// TIA Portal project "BTL_FIX" (V16)

(* hardware
DEVICE "S7300/ET200M station_1"  S7-300 station
   slot 0: "Rail_0"  Rail  6ES7 390-1***0-0AA0
   slot 2: "PLC_1"  CPU 314C-2 PN/DP  6ES7 314-6EH04-0AB0  V3.3
      slot 2: "PROFINET interface_1"  PN-IO
         slot 1: "Port_1"  Port
         slot 2: "Port_2"  Port
      slot 5: "DI 24/DO 16_1"  DI24/DO16
      slot 6: "AI 5/AO 2_1"  AI5/AO2
      slot 7: "Count_1"  Counter
      slot 8: "Positioning_1"  Positioning
   slot 4: "DO 8x24VDC/0.5A_1"  DO8 x 24VDC / 0.5A  6ES7 322-8BF00-0AB0
*)

// ===== PLC "PLC_1"  CPU 314C-2 PN/DP =====

VAR_GLOBAL   // PLC tag table "Default tag table"
   "Tag_1" AT %M100.0 : Bool;
   "Tag_2" AT %M200.0 : Bool;
   "Tag_3" AT %M201.0 : Bool;
END_VAR

VAR_GLOBAL   // PLC tag table "PRO_TAG"
   "Start" AT %I0.0 : Bool;
   "Pause" AT %I0.1 : Bool;
   "EMER" AT %I0.2 : Bool;
   "RESET" AT %I0.3 : Bool;
   "MODE" AT %I0.4 : Bool;
   "HALF_AUTO" AT %I2.6 : Bool;
   "PHOI" AT %I0.5 : Bool;
   "A0" AT %I1.0 : Bool;
   "A1" AT %I1.1 : Bool;
   "B0" AT %I1.2 : Bool;
   "B1" AT %I1.3 : Bool;
   "C0" AT %I1.4 : Bool;
   "C1" AT %I1.5 : Bool;
   "A_FOR" AT %Q0.0 : Bool;
   "A_REV" AT %Q0.1 : Bool;
   "B_FOR" AT %Q0.2 : Bool;
   "B_REV" AT %Q0.3 : Bool;
   "C_FOR" AT %Q0.4 : Bool;
   "C_REV" AT %Q0.5 : Bool;
   "S0" AT %M8.0 : Bool;
   "S1" AT %M8.1 : Bool;
   "S2" AT %M8.2 : Bool;
   "S3" AT %M8.3 : Bool;
   "S4" AT %M8.4 : Bool;
   "S5" AT %M8.5 : Bool;
   "S6" AT %M8.6 : Bool;
   "S7" AT %M8.7 : Bool;
   "S_NULL" AT %M9.0 : Bool;
   "S_EMER" AT %M9.1 : Bool;
   "S_PAUSE" AT %M9.2 : Bool;
   "T01" AT %M3.1 : Bool;
   "T1_PAUSE" AT %M3.2 : Bool;
   "T1_EMER" AT %M3.3 : Bool;
   "T12" AT %M3.4 : Bool;
   "T2_PAUSE" AT %M3.5 : Bool;
   "T2_EMER" AT %M3.6 : Bool;
   "T23" AT %M3.7 : Bool;
   "T3_PAUSE" AT %M4.0 : Bool;
   "T3_EMER" AT %M4.1 : Bool;
   "T34" AT %M4.2 : Bool;
   "T4_PAUSE" AT %M4.3 : Bool;
   "T4_EMER" AT %M4.4 : Bool;
   "T45" AT %M4.5 : Bool;
   "T5_PAUSE" AT %M4.6 : Bool;
   "T5_EMER" AT %M4.7 : Bool;
   "T56" AT %M5.0 : Bool;
   "T6_PAUSE" AT %M5.1 : Bool;
   "T6_EMER" AT %M5.2 : Bool;
   "T67" AT %M5.3 : Bool;
   "T7_PAUSE" AT %M5.4 : Bool;
   "T7_EMER" AT %M5.5 : Bool;
   "T7_NULL" AT %M5.6 : Bool;
   "T_NULL_S1" AT %M5.7 : Bool;
   "T_EMER_RESET" AT %M6.0 : Bool;
   "T_PAUSE_EMER" AT %M6.1 : Bool;
   "T_PAUSE_S1" AT %M6.2 : Bool;
   "T_PAUSE_S2" AT %M6.3 : Bool;
   "T_PAUSE_S3" AT %M6.4 : Bool;
   "T_PAUSE_S4" AT %M6.5 : Bool;
   "T_PAUSE_S5" AT %M6.6 : Bool;
   "T_PAUSE_S6" AT %M6.7 : Bool;
   "T_PAUSE_S7" AT %M7.0 : Bool;
   "T_PAUSE_NULL" AT %M7.1 : Bool;
   "T_NULL_PAUSE" AT %M7.2 : Bool;
   "T_NULL_EMER" AT %M7.3 : Bool;
   "INT_PAUSE" AT %MW10 : Int;
   "T00" AT %M3.0 : Bool;
   "TEMP_START" AT %M7.4 : Bool;
   "Q_START" AT %Q0.6 : Bool;
   "Q_MODE" AT %Q0.7 : Bool;
   "Q_WAIT" AT %Q1.6 : Bool;
   "FIRST_SCAN" AT %M1.7 : Bool;
   "TEMP_FIRST" AT %M2.0 : Bool;
   "S_RESET" AT %M2.1 : Bool;
   "T_RESET_S1" AT %M2.2 : Bool;
   "no_name" AT %M2.3 : Bool;
   "Q_EMER" AT %Q1.7 : Bool;
   "INA_FOR" AT %I2.0 : Bool;
   "INA_REV" AT %I2.1 : Bool;
   "INB_FOR" AT %I2.2 : Bool;
   "INB_REV" AT %I2.3 : Bool;
   "INC_FOR" AT %I2.4 : Bool;
   "INC_REV" AT %I2.5 : Bool;
   "Q_PAUSE" AT %Q1.0 : Bool;
   "HA_FOR" AT %M0.0 : Bool;
   "HA_REV" AT %M0.1 : Bool;
   "HB_FOR" AT %M0.2 : Bool;
   "HB_REV" AT %M0.3 : Bool;
   "HC_FOR" AT %M0.4 : Bool;
   "HC_REV" AT %M0.5 : Bool;
   "Q_PHOI" AT %Q1.1 : Bool;
   "STOP" AT %I0.6 : Bool;
   "TEMP_OFF" AT %M0.6 : Bool;
   "PHOI_MOI" AT %M200.1 : Bool;
   "T_NULL_OFF" AT %M200.2 : Bool;
   "S_OFF" AT %M200.3 : Bool;
   "T_OFF_S1" AT %M200.4 : Bool;
   "L_ERROR_PHOI" AT %Q2.0 : Bool;
   "L_OFF" AT %Q2.1 : Bool;
   "TRIG_MODE" AT %M200.5 : Bool;
   "TMP_TRIG_MODE" AT %M200.6 : Bool;
   "ALARM_AR" AT %Q2.2 : Bool;
   "ALARM_AF" AT %Q2.3 : Bool;
   "ALARM_BR" AT %Q2.4 : Bool;
   "ALARM_BF" AT %Q2.5 : Bool;
   "ALARM_CR" AT %Q2.6 : Bool;
   "ALARM_CF" AT %Q2.7 : Bool;
   "PHOI_NOT_FOUND" AT %M200.7 : Bool;
END_VAR

FUNCTION "Block_1" : Void   // FC1, LAD
{ S7_Optimized_Access := 'FALSE' }
VERSION : 0.1
   VAR_INPUT
      in : Bool;
   END_VAR
   VAR_OUTPUT
      out : Bool;
   END_VAR
   VAR_TEMP   // added for the SCL form of the ladder/FBD networks
      _w1 : Bool;
   END_VAR
BEGIN

REGION Network 1
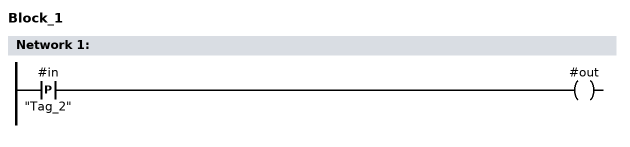
   RUNG wire#powerrail
      P_Contact(operand := #in, bit := "Tag_2")
      Coil( #out )
   END_RUNG
   // the same network as SCL:
   #_w1 := #in AND NOT "Tag_2";   // rising edge of #in
   "Tag_2" := #in;
   #out := #_w1;
END_REGION
END_FUNCTION

FUNCTION "Block_2" : Void   // FC2, LAD
{ S7_Optimized_Access := 'FALSE' }
VERSION : 0.1
   VAR_INPUT
      in : Bool;
   END_VAR
   VAR_OUTPUT
      out : Bool;
   END_VAR
   VAR_TEMP   // added for the SCL form of the ladder/FBD networks
      _w1 : Bool;
   END_VAR
BEGIN

REGION Network 1
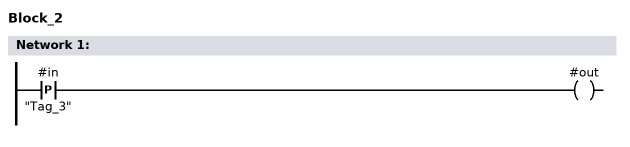
   RUNG wire#powerrail
      P_Contact(operand := #in, bit := "Tag_3")
      Coil( #out )
   END_RUNG
   // the same network as SCL:
   #_w1 := #in AND NOT "Tag_3";   // rising edge of #in
   "Tag_3" := #in;
   #out := #_w1;
END_REGION
END_FUNCTION

ORGANIZATION_BLOCK "Main"   // OB1, SCL
TITLE = "Main Program Sweep (Cycle)"
{ S7_Optimized_Access := 'FALSE' }
VERSION : 0.1
   VAR_TEMP
      OB1_EV_CLASS : Byte;   // Bits 0-3 = 1 (Coming event), Bits 4-7 = 1 (Event class 1)
      OB1_SCAN_1 : Byte;   // 1 (Cold restart scan 1 of OB 1), 3 (Scan 2-n of OB 1)
      OB1_PRIORITY : Byte;   // Priority of OB Execution
      OB1_OB_NUMBR : Byte;   // 1 (Organization block 1, OB1)
      OB1_RESERVED_1 : Byte;   // Reserved for system
      OB1_RESERVED_2 : Byte;   // Reserved for system
      OB1_PREV_CYCLE : Int;   // Cycle time of previous OB1 scan (milliseconds)
      OB1_MIN_CYCLE : Int;   // Minimum cycle time of OB1 (milliseconds)
      OB1_MAX_CYCLE : Int;   // Maximum cycle time of OB1 (milliseconds)
      OB1_DATE_TIME : Date_And_Time;   // Date and time OB1 started
   END_VAR
BEGIN
   "IEC_Timer_0_DB".TON(IN:="S_NULL",
                        PT:=T#1S);
   "IEC_Timer_0_DB_1".TOF(IN:="PHOI_MOI",
                          PT:=t#2s);

   IF "STOP" AND NOT "S_EMER" AND NOT "EMER" THEN
       "TEMP_OFF" := 1;
   END_IF;
   IF "TEMP_OFF" AND "Start" THEN
       "TEMP_OFF" := 0;
   END_IF;

   IF NOT "S_EMER" THEN
       "Block_1"(in := "MODE",
                 out => "TRIG_MODE");
   END_IF;
   "Block_2"(in:="PHOI",
             out=>"PHOI_MOI");

   REGION
       "Q_MODE" := "MODE";
       "Q_START" := "TEMP_START" AND NOT "S_EMER";
       "Q_WAIT" := "S_NULL" AND NOT "TEMP_OFF" AND "MODE";
       "Q_EMER" := "S_EMER" OR "EMER";
       "Q_PAUSE" := "S_PAUSE" AND NOT "TEMP_START";
       "Q_PHOI" := "PHOI";
       "L_OFF" := "TEMP_OFF";
   END_REGION

   IF NOT "TEMP_FIRST" AND NOT "IEC_Timer_0_DB_2".Q THEN
       "FIRST_SCAN" := 1;
   ELSE
       "FIRST_SCAN" := 0;
   END_IF;

   "IEC_Timer_0_DB_2".TON(IN := "FIRST_SCAN" ,
                          PT := T#2S);

   IF "S0" THEN
       "INT_PAUSE" := 0;
   ELSIF "S1" THEN
       "INT_PAUSE" := 1;
   ELSIF "S2" THEN
       "INT_PAUSE" := 2;
   ELSIF "S3" THEN
       "INT_PAUSE" := 3;
   ELSIF "S4" THEN
       "INT_PAUSE" := 4;
   ELSIF "S5" THEN
       "INT_PAUSE" := 5;
   ELSIF "S6" THEN
       "INT_PAUSE" := 6;
   ELSIF "S7" THEN
       "INT_PAUSE" := 7;
   ELSIF "S_NULL" THEN
       "INT_PAUSE" := 8;
   ELSIF "S_EMER" THEN
       "INT_PAUSE" := 9;

   END_IF;
   "PHOI_NOT_FOUND" := NOT "PHOI" AND "MODE" AND ("S0" OR "S1" OR "S2" OR "S3" OR "S4" OR "S5" OR "S6" OR "S7" OR "S_EMER" OR "S_RESET" OR "S_PAUSE");

   IF "MODE" THEN // CHE DO TU DONG

       IF ("Start" AND NOT "Pause" AND "PHOI" AND NOT "TRIG_MODE" AND NOT "S_EMER" AND NOT "S_RESET") THEN
           "TEMP_START" := 1;
       ELSIF (NOT "Start" AND "Pause") OR "S_EMER" THEN
           "TEMP_START" := 0;
       END_IF;
       // TRANSITION LOGIC
       "T00" := "FIRST_SCAN";
       "T01" := "S0" AND "TEMP_START" AND "PHOI";
       "T12" := "S1" AND "A1";
       "T23" := "S2" AND "B1";
       "T34" := "S3" AND "B0";
       "T45" := "S4" AND "C1";
       "T56" := "S5" AND "B1";
       "T67" := "S6" AND "B0";
       "T7_NULL" := "S7" AND "A0" AND "C0";
       "T_NULL_S1" := "S_NULL" AND "PHOI_MOI" AND "IEC_Timer_0_DB".Q AND NOT "TEMP_OFF";
       "T_NULL_OFF" := "S_NULL" AND "TEMP_OFF";
       "T_OFF_S1" := "S_OFF" AND "TEMP_START" AND "PHOI";

       "T1_EMER" := "S1" AND ("EMER" OR "TRIG_MODE" OR "PHOI_NOT_FOUND");
       "T2_EMER" := "S2" AND ("EMER" OR "TRIG_MODE" OR "PHOI_NOT_FOUND");
       "T3_EMER" := "S3" AND ("EMER" OR "TRIG_MODE" OR "PHOI_NOT_FOUND");
       "T4_EMER" := "S4" AND ("EMER" OR "TRIG_MODE" OR "PHOI_NOT_FOUND");
       "T5_EMER" := "S5" AND ("EMER" OR "TRIG_MODE" OR "PHOI_NOT_FOUND");
       "T6_EMER" := "S6" AND ("EMER" OR "TRIG_MODE" OR "PHOI_NOT_FOUND");
       "T7_EMER" := "S7" AND ("EMER" OR "TRIG_MODE" OR "PHOI_NOT_FOUND");
       "T_NULL_EMER" := "S_NULL" AND ("EMER" OR "TRIG_MODE" OR "PHOI_NOT_FOUND");
       "T_PAUSE_EMER" := "S_PAUSE" AND ("EMER" OR "TRIG_MODE" OR "PHOI_NOT_FOUND");

       "T1_PAUSE" := "S1" AND "Pause";
       "T2_PAUSE" := "S2" AND "Pause";
       "T3_PAUSE" := "S3" AND "Pause";
       "T4_PAUSE" := "S4" AND "Pause";
       "T5_PAUSE" := "S5" AND "Pause";
       "T6_PAUSE" := "S6" AND "Pause";
       "T7_PAUSE" := "S7" AND "Pause";
       "T_NULL_PAUSE" := "S_NULL" AND "Pause";

       "T_EMER_RESET" := "S_EMER" AND ("RESET" OR "TMP_TRIG_MODE");
       "T_RESET_S1" := "S_RESET" AND "A0" AND "B0" AND "C0" ;

       "T_PAUSE_S1" := "S_PAUSE" AND "Start" AND ("INT_PAUSE" = 1);
       "T_PAUSE_S2" := "S_PAUSE" AND "Start" AND ("INT_PAUSE" = 2);
       "T_PAUSE_S3" := "S_PAUSE" AND "Start" AND ("INT_PAUSE" = 3);
       "T_PAUSE_S4" := "S_PAUSE" AND "Start" AND ("INT_PAUSE" = 4);
       "T_PAUSE_S5" := "S_PAUSE" AND "Start" AND ("INT_PAUSE" = 5);
       "T_PAUSE_S6" := "S_PAUSE" AND "Start" AND ("INT_PAUSE" = 6);
       "T_PAUSE_S7" := "S_PAUSE" AND "Start" AND ("INT_PAUSE" = 7);
       "T_PAUSE_NULL" := "S_PAUSE" AND "Start" AND ("INT_PAUSE" = 8);


       // STATE LOGIC 
       "S0" := ("S0" OR "T00") AND NOT "S_OFF" AND NOT "T01" AND NOT "S1" AND NOT "S2" AND NOT "S3" AND NOT "S4" AND NOT "S5" AND NOT "S6" AND NOT "S7" AND NOT "S_NULL" AND NOT "S_PAUSE" AND NOT "S_EMER" AND NOT "S_RESET";
       "S1" := ("S1" OR "T01" OR "T_PAUSE_S1" OR "T_NULL_S1" OR 0 OR "T_OFF_S1" ) AND NOT"T12" AND NOT "T1_PAUSE" AND NOT "T1_EMER" AND NOT "IEC_Timer_0_DB_1".Q;
       "S2" := ("S2" OR "T12" OR "T_PAUSE_S2") AND NOT "T23" AND NOT "T2_PAUSE" AND NOT "T2_EMER";
       "S3" := ("S3" OR "T23" OR "T_PAUSE_S3") AND NOT "T34" AND NOT "T3_PAUSE" AND NOT "T3_EMER";
       "S4" := ("S4" OR "T34" OR "T_PAUSE_S4") AND NOT "T45" AND NOT "T4_PAUSE" AND NOT "T4_EMER";
       "S5" := ("S5" OR "T45" OR "T_PAUSE_S5") AND NOT "T56" AND NOT "T5_PAUSE" AND NOT "T5_EMER";
       "S6" := ("S6" OR "T56" OR "T_PAUSE_S6") AND NOT "T67" AND NOT "T6_PAUSE" AND NOT "T6_EMER";
       "S7" := ("S7" OR "T67" OR "T_PAUSE_S7") AND NOT "T7_NULL" AND NOT "T7_PAUSE" AND NOT "T7_EMER";
       "S_NULL" := ("S_NULL" OR "T7_NULL" OR "T_PAUSE_NULL" OR "T_RESET_S1") AND NOT "T_NULL_EMER" AND NOT "T_NULL_S1" AND NOT "T_NULL_PAUSE" AND NOT "T_NULL_OFF";
       "S_PAUSE" := ("S_PAUSE" OR "T1_PAUSE" OR "T2_PAUSE" OR "T3_PAUSE" OR "T4_PAUSE" OR "T5_PAUSE" OR "T6_PAUSE" OR "T7_PAUSE" OR "T_NULL_PAUSE") AND NOT "T_PAUSE_S1" AND NOT "T_PAUSE_S2" AND NOT "T_PAUSE_S3" AND NOT "T_PAUSE_S4" AND NOT "T_PAUSE_S5" AND NOT "T_PAUSE_S6" AND NOT "T_PAUSE_S7" AND NOT "T_PAUSE_NULL" AND NOT "T_PAUSE_EMER";
       "S_EMER" := "EMER" OR ("S_EMER" OR "T1_EMER" OR "T2_EMER" OR "T3_EMER" OR "T4_EMER" OR "T5_EMER" OR "T6_EMER" OR "T7_EMER" OR "T_NULL_EMER" OR "T_PAUSE_EMER") AND NOT "T_EMER_RESET";
       "S_RESET" := ("S_RESET" OR "T_EMER_RESET") AND NOT "T_RESET_S1";
       "S_OFF" := ("S_OFF" OR "T_NULL_OFF") AND NOT "T_OFF_S1";

   ELSIF NOT "MODE" THEN  // CHE DO CHINH TAY 
       IF ("Start" AND NOT "Pause") THEN
           "TEMP_START" := 1;
       ELSIF (NOT "Start" AND "Pause") OR "S_EMER" THEN
           "TEMP_START" := 0;
       END_IF;

       IF "EMER" THEN
           "TEMP_START" := 0;
       END_IF;

       IF NOT "S_EMER" AND NOT "EMER" AND "TEMP_START" AND NOT "HALF_AUTO" THEN
           "A_FOR" := "INA_FOR" AND NOT "A1";
           "A_REV" := "INA_REV" AND NOT "A0";
           "B_FOR" := "INB_FOR" AND NOT "B1";
           "B_REV" := "INB_REV" AND NOT "B0";
           "C_FOR" := "INC_FOR" AND NOT "C1" AND NOT "B1";
           "C_REV" := "INC_REV" AND NOT "C0" AND NOT "B1";
       ELSIF NOT "S_EMER" AND NOT "EMER"  AND "HALF_AUTO" THEN
           IF "INA_FOR" AND NOT "HA_REV" AND "TEMP_START" AND "A0" THEN
               "HA_FOR" := 1;
           ELSIF (NOT "INA_FOR" AND "A1") OR "Pause" THEN
               "HA_FOR" := 0;
           END_IF;
           IF "INA_REV" AND NOT "HA_FOR" AND "TEMP_START" THEN
               "HA_REV" := 1;
           ELSIF (NOT "INA_REV" AND "A0") OR "Pause" THEN
               "HA_REV" := 0;
           END_IF;
           "A_FOR" := "HA_FOR" AND "TEMP_START" AND NOT "EMER" AND NOT "S_EMER";
           "A_REV" := "HA_REV" AND "TEMP_START" AND NOT "EMER" AND NOT "S_EMER";

           IF "INB_FOR" AND NOT "HB_REV" AND "TEMP_START" AND "B0" AND NOT "C_FOR" AND NOT "C_REV" THEN
               "HB_FOR" := 1;
           ELSIF (NOT "INB_FOR" AND "B1") OR "Pause" THEN
               "HB_FOR" := 0;
           END_IF;
           IF "INB_REV" AND NOT "HB_FOR" AND "TEMP_START" AND NOT "C_FOR" AND NOT "C_REV" THEN
               "HB_REV" := 1;
           ELSIF (NOT "INB_REV" AND "B0") OR "Pause" THEN
               "HB_REV" := 0;
           END_IF;
           "B_FOR" := "HB_FOR" AND "TEMP_START" AND NOT "EMER" AND NOT "S_EMER";
           "B_REV" := "HB_REV" AND "TEMP_START" AND NOT "EMER" AND NOT "S_EMER";
           IF "INC_FOR" AND NOT "HC_REV" AND "TEMP_START" AND "C0" AND "B0" THEN
               "HC_FOR" := 1;
           ELSIF (NOT "INC_FOR" AND "C1") OR "Pause"  THEN
               "HC_FOR" := 0;
           END_IF;
           IF "INC_REV" AND NOT "HC_FOR" AND "TEMP_START" AND "B0" THEN
               "HC_REV" := 1;
           ELSIF (NOT "INC_REV" AND "C0") OR "Pause" THEN
               "HC_REV" := 0;
           END_IF;
           "C_FOR" := "HC_FOR" AND "TEMP_START" AND NOT "EMER" AND NOT "S_EMER";
           "C_REV" := "HC_REV" AND "TEMP_START" AND NOT "EMER" AND NOT "S_EMER";

       END_IF;
   END_IF;


   IF "S_EMER" AND "TRIG_MODE" AND NOT "EMER" THEN
       "TMP_TRIG_MODE" := 1;
   ELSE
       "TMP_TRIG_MODE" := 0;
   END_IF;

   // OUTPUT 
   IF "TEMP_START" AND "MODE" AND "PHOI" AND NOT "TRIG_MODE" THEN
       "A_FOR" := "S1" AND NOT "A1";
       "A_REV" := "S7" AND NOT "A0";
       "B_FOR" := ("S2" OR "S5") AND NOT "B1";
       "B_REV" := ("S3" OR "S6") AND NOT "B0";
       "C_FOR" := "S4" AND NOT "C1";
       "C_REV" := "S7" AND NOT "C0";
       "L_ERROR_PHOI" := 0;
   ELSIF "TEMP_START" AND "MODE" AND NOT "PHOI" AND NOT "TRIG_MODE" THEN
       "L_ERROR_PHOI" := NOT "S_NULL";
       "A_FOR" := 0;
       "A_REV" := 0;
       "B_FOR" := 0;
       "B_REV" := 0;
       "C_FOR" := 0;
       "C_REV" := 0;
   ELSIF NOT "TEMP_START" AND "MODE" AND NOT "TRIG_MODE" THEN
       "A_FOR" := 0;
       "A_REV" := 0;
       "B_FOR" := 0;
       "B_REV" := 0;
       "C_FOR" := 0;
       "C_REV" := 0;
   END_IF;
   IF "S_RESET" AND "MODE" THEN
       "A_REV" := NOT "A0" AND "B0";
       "B_REV" := NOT "B0";
       "C_REV" := NOT "C0" AND "B0";
   END_IF;
   IF "EMER" OR "S_EMER" THEN
       "A_FOR" := 0;
       "A_REV" := 0;
       "B_FOR" := 0;
       "B_REV" := 0;
       "C_FOR" := 0;
       "C_REV" := 0;
   END_IF;
   IF "S_OFF" THEN
       "TEMP_START" := 0;
       "TEMP_OFF" := 0;
       "A_FOR" := 0;
       "A_REV" := NOT "A0" AND "B0";
       "B_FOR" := 0;
       "B_REV" := NOT "B0";
       "C_FOR" := 0;
       "C_REV" := NOT "C0" AND "B0";
   END_IF;
   REGION ALARM

       "CHECK_AREV".TON(IN := "A_REV" AND NOT "A0",
                        PT := T#10S,
                        Q => "ALARM_AR");
       "CHECK_AFOR".TON(IN := "A_FOR" AND NOT "A1",
                        PT := T#10S,
                        Q => "ALARM_AF");
       "CHECK_BREV".TON(IN := "B_REV" AND NOT "B0",
                        PT := T#10S,
                        Q => "ALARM_BR");
       "CHECK_BFOR".TON(IN := "B_FOR" AND NOT "B1",
                        PT := T#10S,
                        Q => "ALARM_BF");
       "CHECK_CREV".TON(IN := "C_REV" AND NOT "C0",
                        PT := T#10S,
                        Q => "ALARM_CR");
       "CHECK_CFOR".TON(IN := "C_FOR" AND NOT "C1",
                        PT := T#10S,
                        Q => "ALARM_CF");
   END_REGION
END_ORGANIZATION_BLOCK

ORGANIZATION_BLOCK "COMPLETE RESTART"   // OB100, LAD
TITLE = "Complete Restart"
{ S7_Optimized_Access := 'FALSE' }
VERSION : 0.1
   VAR_TEMP
      OB100_EV_CLASS : Byte;   // 16#13, Event class 1, Entering event state, Event logged in diagnostic buffer
      OB100_STRTUP : Byte;   // 16#81/82/83/84 Method of startup
      OB100_PRIORITY : Byte;   // Priority of OB Execution
      OB100_OB_NUMBR : Byte;   // 100 (Organization block 100, OB100)
      OB100_RESERVED_1 : Byte;   // Reserved for system
      OB100_RESERVED_2 : Byte;   // Reserved for system
      OB100_STOP : Word;   // Event that caused CPU to stop (16#4xxx)
      OB100_STRT_INFO : DWord;   // Information on how system started
      OB100_DATE_TIME : Date_And_Time;   // Date and time OB100 started
   END_VAR
BEGIN

REGION Network 1
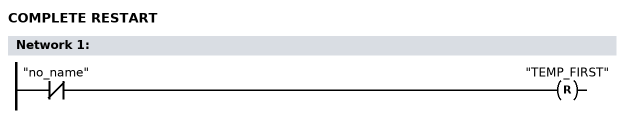
   RUNG wire#powerrail
      I_Contact( "no_name" )
      R_Coil( "TEMP_FIRST" )
   END_RUNG
   // the same network as SCL:
   IF NOT "no_name" THEN "TEMP_FIRST" := FALSE; END_IF;
END_REGION
END_ORGANIZATION_BLOCK